Universal Robots PolyScope program: show_gripper.urp

Program show_gripper (installation=default directory=/programs createdIn=5.9.1.1031110 lastSavedIn=5.9.1.1031110 robotSerialNumber=20195501059)
Calibrated DH parameters: a=[0.000146, -0.418764, -0.053981, 0.000058, -0.000023, 0]; d=[0.162545, 37.319448, -206.067439, 168.881546, 0.09955, 0.099464]; alpha=[1.57004, -0.001979, 0.002304, 1.570607, -1.57066, 0]; deltaTheta=[0, -0.174616, -1.258233, 1.432844, -0.000001, 0]
Robot Program (runOnlyOnce=false)
  Call ShowGripper
SubProgram -> ShowGripper
SubProgram ShowGripper (keepSynchronizedWithDisk=false)
  MoveJ speed 60 deg/s, acceleration 80 deg/s^2 (useActiveTCP=true) feature=Base
    Waypoint Waypoint_1: TCP in base x=1021.007 y=-270.578 z=147.215 mm, rx=0.3291 ry=1.7401 rz=-0.2274 rad; joints [157.047, -16.074, 43.041, -195.788, 273.242, 91.023] deg; TCP offset x=0 y=0 z=174 mm, rx=0 ry=0 rz=0 rad
